{attribute 'qualified_only'}
VAR_GLOBAL CONSTANT
	cEventClassNameLength : UDINT (80..255) := 80;
	cMessageTextLength : UDINT(80..1024) := 255;
	cSourceNameLength : UDINT (80..255) := 80;
	cMaxConcurrentEvents : UDINT (1..64) := 16;
	cMaxJsonTextLength : UDINT (80..16384) := 1024;
END_VAR

(* stored: Version 1.1.0.1, ProductVersion 3.1.4024.12
   GVL Param_EventLoggerListener: Id {2aac157d-e414-4f13-a6ad-dc7028dfe748}, ParameterList True *)
